REGION Network 40: *************** Alarms estop robots ***************
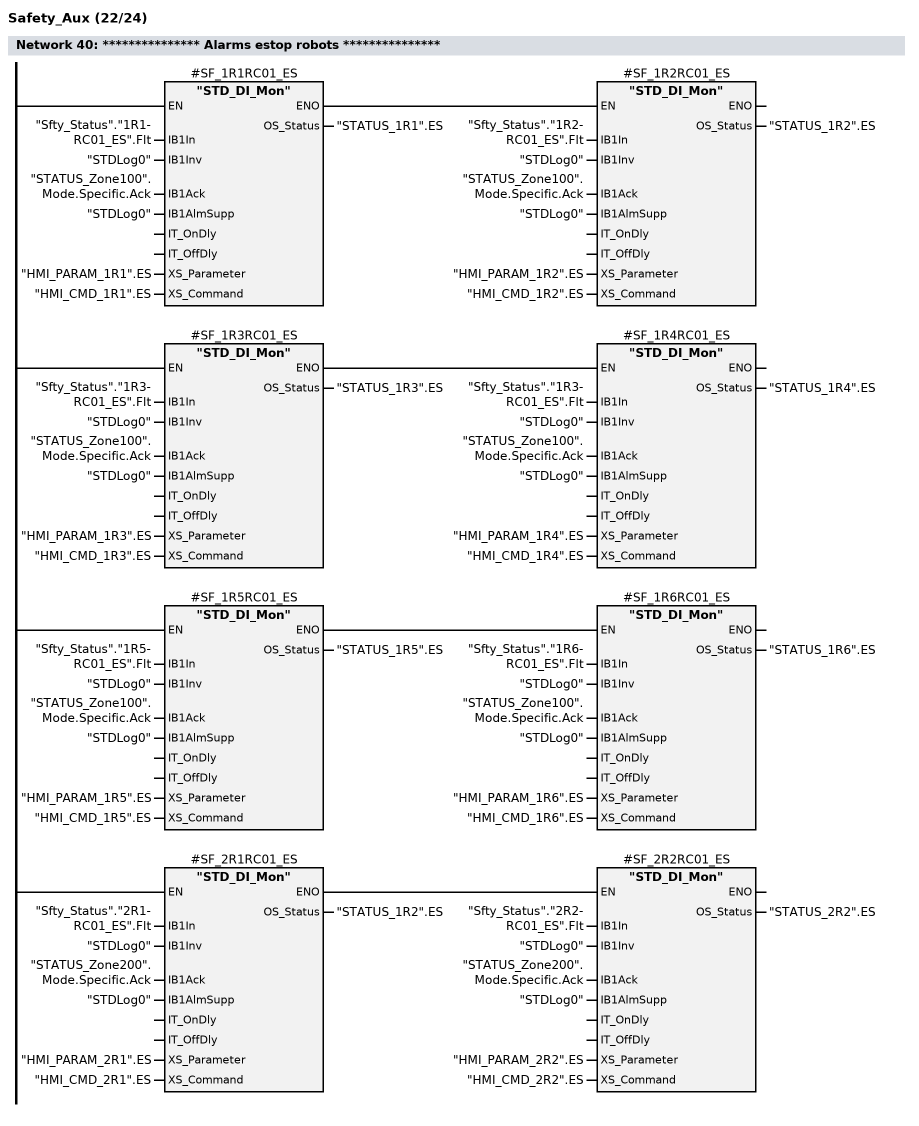
   RUNG wire#powerrail
      #SF_1R1RC01_ES(IB1In := "Sfty_Status"."1R1-RC01_ES".Flt, IB1Inv := "STDLog0", IB1Ack := "STATUS_Zone100".Mode.Specific.Ack, IB1AlmSupp := "STDLog0", IT_OnDly :=, IT_OffDly :=, XS_Parameter := "HMI_PARAM_1R1".ES, XS_Command := "HMI_CMD_1R1".ES, OS_Status => "STATUS_1R1".ES)
      #SF_1R2RC01_ES(IB1In := "Sfty_Status"."1R2-RC01_ES".Flt, IB1Inv := "STDLog0", IB1Ack := "STATUS_Zone100".Mode.Specific.Ack, IB1AlmSupp := "STDLog0", IT_OnDly :=, IT_OffDly :=, XS_Parameter := "HMI_PARAM_1R2".ES, XS_Command := "HMI_CMD_1R2".ES, OS_Status => "STATUS_1R2".ES)
   END_RUNG
   RUNG wire#powerrail
      #SF_1R3RC01_ES(IB1In := "Sfty_Status"."1R3-RC01_ES".Flt, IB1Inv := "STDLog0", IB1Ack := "STATUS_Zone100".Mode.Specific.Ack, IB1AlmSupp := "STDLog0", IT_OnDly :=, IT_OffDly :=, XS_Parameter := "HMI_PARAM_1R3".ES, XS_Command := "HMI_CMD_1R3".ES, OS_Status => "STATUS_1R3".ES)
      #SF_1R4RC01_ES(IB1In := "Sfty_Status"."1R3-RC01_ES".Flt, IB1Inv := "STDLog0", IB1Ack := "STATUS_Zone100".Mode.Specific.Ack, IB1AlmSupp := "STDLog0", IT_OnDly :=, IT_OffDly :=, XS_Parameter := "HMI_PARAM_1R4".ES, XS_Command := "HMI_CMD_1R4".ES, OS_Status => "STATUS_1R4".ES)
   END_RUNG
   RUNG wire#powerrail
      #SF_1R5RC01_ES(IB1In := "Sfty_Status"."1R5-RC01_ES".Flt, IB1Inv := "STDLog0", IB1Ack := "STATUS_Zone100".Mode.Specific.Ack, IB1AlmSupp := "STDLog0", IT_OnDly :=, IT_OffDly :=, XS_Parameter := "HMI_PARAM_1R5".ES, XS_Command := "HMI_CMD_1R5".ES, OS_Status => "STATUS_1R5".ES)
      #SF_1R6RC01_ES(IB1In := "Sfty_Status"."1R6-RC01_ES".Flt, IB1Inv := "STDLog0", IB1Ack := "STATUS_Zone100".Mode.Specific.Ack, IB1AlmSupp := "STDLog0", IT_OnDly :=, IT_OffDly :=, XS_Parameter := "HMI_PARAM_1R6".ES, XS_Command := "HMI_CMD_1R6".ES, OS_Status => "STATUS_1R6".ES)
   END_RUNG
   RUNG wire#powerrail
      #SF_2R1RC01_ES(IB1In := "Sfty_Status"."2R1-RC01_ES".Flt, IB1Inv := "STDLog0", IB1Ack := "STATUS_Zone200".Mode.Specific.Ack, IB1AlmSupp := "STDLog0", IT_OnDly :=, IT_OffDly :=, XS_Parameter := "HMI_PARAM_2R1".ES, XS_Command := "HMI_CMD_2R1".ES, OS_Status => "STATUS_1R2".ES)
      #SF_2R2RC01_ES(IB1In := "Sfty_Status"."2R2-RC01_ES".Flt, IB1Inv := "STDLog0", IB1Ack := "STATUS_Zone200".Mode.Specific.Ack, IB1AlmSupp := "STDLog0", IT_OnDly :=, IT_OffDly :=, XS_Parameter := "HMI_PARAM_2R2".ES, XS_Command := "HMI_CMD_2R2".ES, OS_Status => "STATUS_2R2".ES)
   END_RUNG
   // the same network as SCL:
   #SF_1R1RC01_ES(IB1In := "Sfty_Status"."1R1-RC01_ES".Flt,   // "STD_DI_Mon"
                  IB1Inv := "STDLog0",
                  IB1Ack := "STATUS_Zone100".Mode.Specific.Ack,
                  IB1AlmSupp := "STDLog0",
                  XS_Parameter := "HMI_PARAM_1R1".ES,
                  XS_Command := "HMI_CMD_1R1".ES,
                  OS_Status => "STATUS_1R1".ES,
                  ENO => #_w1);
   IF #_w1 THEN
       #SF_1R2RC01_ES(IB1In := "Sfty_Status"."1R2-RC01_ES".Flt,   // "STD_DI_Mon"
                      IB1Inv := "STDLog0",
                      IB1Ack := "STATUS_Zone100".Mode.Specific.Ack,
                      IB1AlmSupp := "STDLog0",
                      XS_Parameter := "HMI_PARAM_1R2".ES,
                      XS_Command := "HMI_CMD_1R2".ES,
                      OS_Status => "STATUS_1R2".ES);
   END_IF;
   #SF_1R3RC01_ES(IB1In := "Sfty_Status"."1R3-RC01_ES".Flt,   // "STD_DI_Mon"
                  IB1Inv := "STDLog0",
                  IB1Ack := "STATUS_Zone100".Mode.Specific.Ack,
                  IB1AlmSupp := "STDLog0",
                  XS_Parameter := "HMI_PARAM_1R3".ES,
                  XS_Command := "HMI_CMD_1R3".ES,
                  OS_Status => "STATUS_1R3".ES,
                  ENO => #_w2);
   IF #_w2 THEN
       #SF_1R4RC01_ES(IB1In := "Sfty_Status"."1R3-RC01_ES".Flt,   // "STD_DI_Mon"
                      IB1Inv := "STDLog0",
                      IB1Ack := "STATUS_Zone100".Mode.Specific.Ack,
                      IB1AlmSupp := "STDLog0",
                      XS_Parameter := "HMI_PARAM_1R4".ES,
                      XS_Command := "HMI_CMD_1R4".ES,
                      OS_Status => "STATUS_1R4".ES);
   END_IF;
   #SF_1R5RC01_ES(IB1In := "Sfty_Status"."1R5-RC01_ES".Flt,   // "STD_DI_Mon"
                  IB1Inv := "STDLog0",
                  IB1Ack := "STATUS_Zone100".Mode.Specific.Ack,
                  IB1AlmSupp := "STDLog0",
                  XS_Parameter := "HMI_PARAM_1R5".ES,
                  XS_Command := "HMI_CMD_1R5".ES,
                  OS_Status => "STATUS_1R5".ES,
                  ENO => #_w3);
   IF #_w3 THEN
       #SF_1R6RC01_ES(IB1In := "Sfty_Status"."1R6-RC01_ES".Flt,   // "STD_DI_Mon"
                      IB1Inv := "STDLog0",
                      IB1Ack := "STATUS_Zone100".Mode.Specific.Ack,
                      IB1AlmSupp := "STDLog0",
                      XS_Parameter := "HMI_PARAM_1R6".ES,
                      XS_Command := "HMI_CMD_1R6".ES,
                      OS_Status => "STATUS_1R6".ES);
   END_IF;
   #SF_2R1RC01_ES(IB1In := "Sfty_Status"."2R1-RC01_ES".Flt,   // "STD_DI_Mon"
                  IB1Inv := "STDLog0",
                  IB1Ack := "STATUS_Zone200".Mode.Specific.Ack,
                  IB1AlmSupp := "STDLog0",
                  XS_Parameter := "HMI_PARAM_2R1".ES,
                  XS_Command := "HMI_CMD_2R1".ES,
                  OS_Status => "STATUS_1R2".ES,
                  ENO => #_w4);
   IF #_w4 THEN
       #SF_2R2RC01_ES(IB1In := "Sfty_Status"."2R2-RC01_ES".Flt,   // "STD_DI_Mon"
                      IB1Inv := "STDLog0",
                      IB1Ack := "STATUS_Zone200".Mode.Specific.Ack,
                      IB1AlmSupp := "STDLog0",
                      XS_Parameter := "HMI_PARAM_2R2".ES,
                      XS_Command := "HMI_CMD_2R2".ES,
                      OS_Status => "STATUS_2R2".ES);
   END_IF;
END_REGION

REGION Network 41: *************** Alarms modules ***************
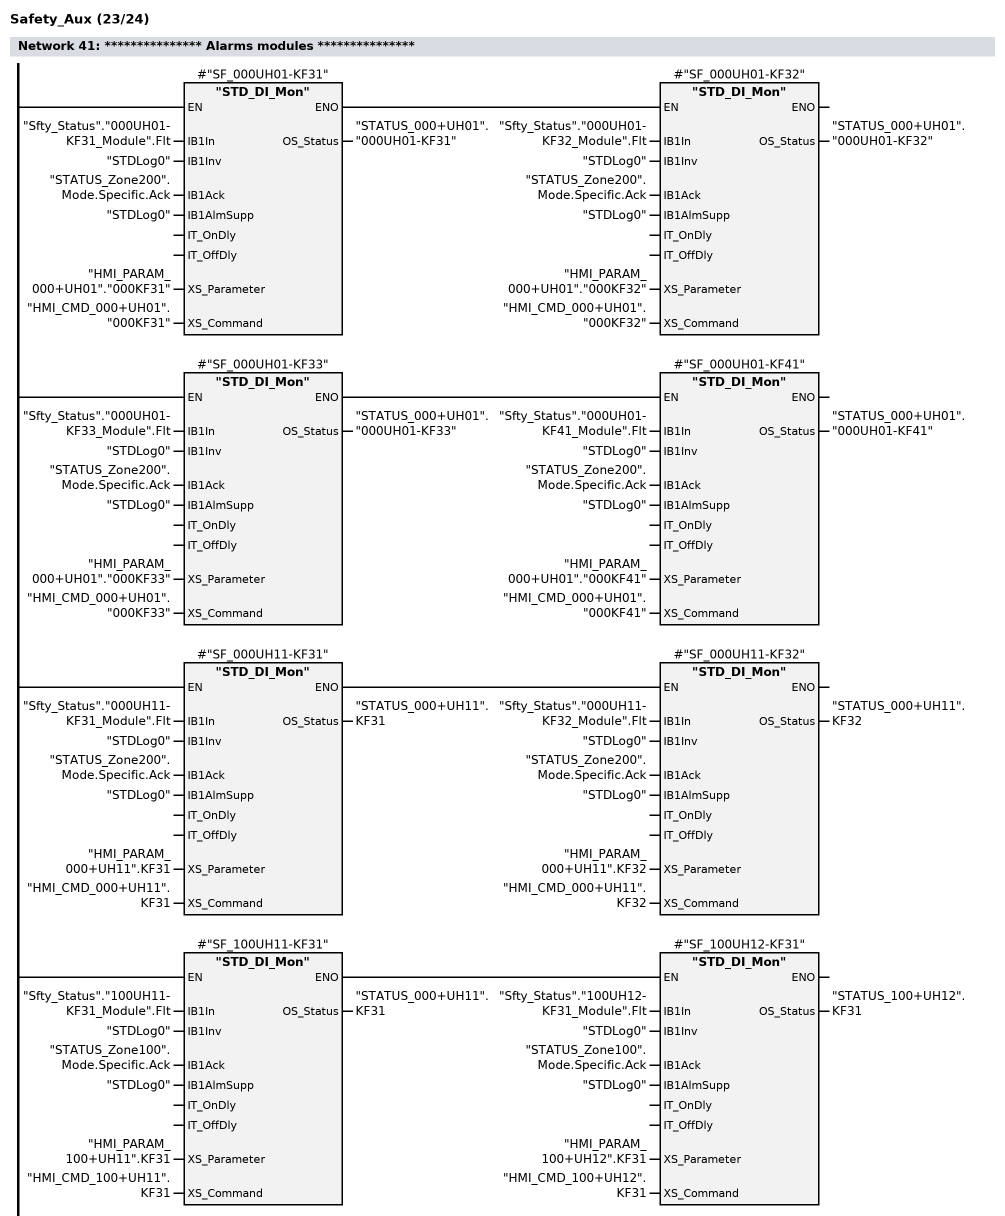
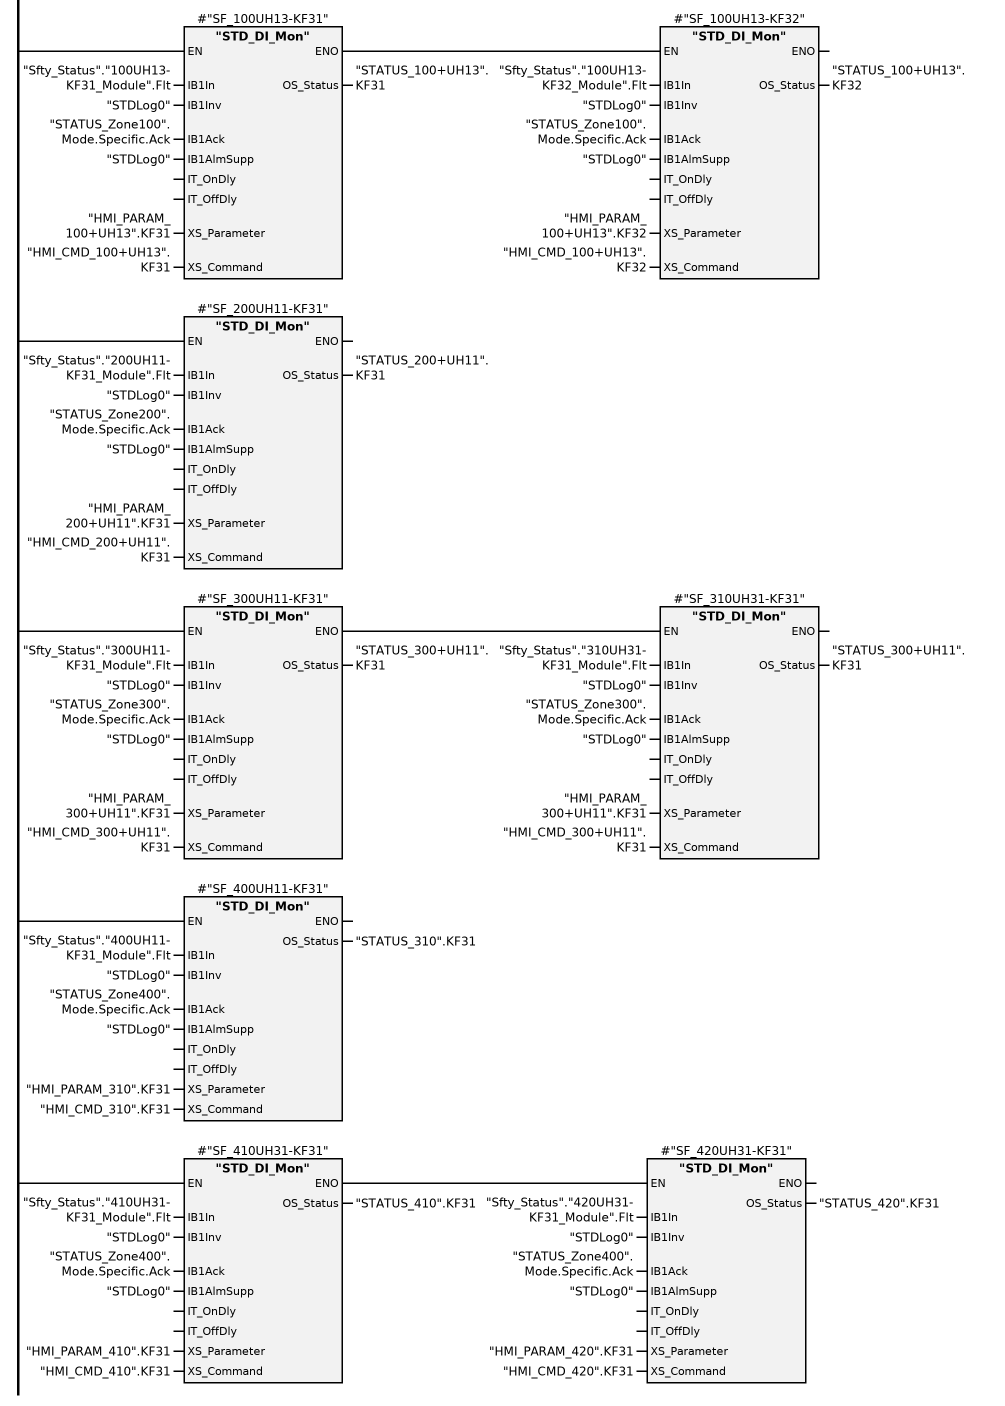
   RUNG wire#powerrail
      #"SF_000UH01-KF31"(IB1In := "Sfty_Status"."000UH01-KF31_Module".Flt, IB1Inv := "STDLog0", IB1Ack := "STATUS_Zone200".Mode.Specific.Ack, IB1AlmSupp := "STDLog0", IT_OnDly :=, IT_OffDly :=, XS_Parameter := "HMI_PARAM_000+UH01"."000KF31", XS_Command := "HMI_CMD_000+UH01"."000KF31", OS_Status => "STATUS_000+UH01"."000UH01-KF31")
      #"SF_000UH01-KF32"(IB1In := "Sfty_Status"."000UH01-KF32_Module".Flt, IB1Inv := "STDLog0", IB1Ack := "STATUS_Zone200".Mode.Specific.Ack, IB1AlmSupp := "STDLog0", IT_OnDly :=, IT_OffDly :=, XS_Parameter := "HMI_PARAM_000+UH01"."000KF32", XS_Command := "HMI_CMD_000+UH01"."000KF32", OS_Status => "STATUS_000+UH01"."000UH01-KF32")
   END_RUNG
   RUNG wire#powerrail
      #"SF_000UH01-KF33"(IB1In := "Sfty_Status"."000UH01-KF33_Module".Flt, IB1Inv := "STDLog0", IB1Ack := "STATUS_Zone200".Mode.Specific.Ack, IB1AlmSupp := "STDLog0", IT_OnDly :=, IT_OffDly :=, XS_Parameter := "HMI_PARAM_000+UH01"."000KF33", XS_Command := "HMI_CMD_000+UH01"."000KF33", OS_Status => "STATUS_000+UH01"."000UH01-KF33")
      #"SF_000UH01-KF41"(IB1In := "Sfty_Status"."000UH01-KF41_Module".Flt, IB1Inv := "STDLog0", IB1Ack := "STATUS_Zone200".Mode.Specific.Ack, IB1AlmSupp := "STDLog0", IT_OnDly :=, IT_OffDly :=, XS_Parameter := "HMI_PARAM_000+UH01"."000KF41", XS_Command := "HMI_CMD_000+UH01"."000KF41", OS_Status => "STATUS_000+UH01"."000UH01-KF41")
   END_RUNG
   RUNG wire#powerrail
      #"SF_000UH11-KF31"(IB1In := "Sfty_Status"."000UH11-KF31_Module".Flt, IB1Inv := "STDLog0", IB1Ack := "STATUS_Zone200".Mode.Specific.Ack, IB1AlmSupp := "STDLog0", IT_OnDly :=, IT_OffDly :=, XS_Parameter := "HMI_PARAM_000+UH11".KF31, XS_Command := "HMI_CMD_000+UH11".KF31, OS_Status => "STATUS_000+UH11".KF31)
      #"SF_000UH11-KF32"(IB1In := "Sfty_Status"."000UH11-KF32_Module".Flt, IB1Inv := "STDLog0", IB1Ack := "STATUS_Zone200".Mode.Specific.Ack, IB1AlmSupp := "STDLog0", IT_OnDly :=, IT_OffDly :=, XS_Parameter := "HMI_PARAM_000+UH11".KF32, XS_Command := "HMI_CMD_000+UH11".KF32, OS_Status => "STATUS_000+UH11".KF32)
   END_RUNG
   RUNG wire#powerrail
      #"SF_100UH11-KF31"(IB1In := "Sfty_Status"."100UH11-KF31_Module".Flt, IB1Inv := "STDLog0", IB1Ack := "STATUS_Zone100".Mode.Specific.Ack, IB1AlmSupp := "STDLog0", IT_OnDly :=, IT_OffDly :=, XS_Parameter := "HMI_PARAM_100+UH11".KF31, XS_Command := "HMI_CMD_100+UH11".KF31, OS_Status => "STATUS_000+UH11".KF31)
      #"SF_100UH12-KF31"(IB1In := "Sfty_Status"."100UH12-KF31_Module".Flt, IB1Inv := "STDLog0", IB1Ack := "STATUS_Zone100".Mode.Specific.Ack, IB1AlmSupp := "STDLog0", IT_OnDly :=, IT_OffDly :=, XS_Parameter := "HMI_PARAM_100+UH12".KF31, XS_Command := "HMI_CMD_100+UH12".KF31, OS_Status => "STATUS_100+UH12".KF31)
   END_RUNG
   RUNG wire#powerrail
      #"SF_100UH13-KF31"(IB1In := "Sfty_Status"."100UH13-KF31_Module".Flt, IB1Inv := "STDLog0", IB1Ack := "STATUS_Zone100".Mode.Specific.Ack, IB1AlmSupp := "STDLog0", IT_OnDly :=, IT_OffDly :=, XS_Parameter := "HMI_PARAM_100+UH13".KF31, XS_Command := "HMI_CMD_100+UH13".KF31, OS_Status => "STATUS_100+UH13".KF31)
      #"SF_100UH13-KF32"(IB1In := "Sfty_Status"."100UH13-KF32_Module".Flt, IB1Inv := "STDLog0", IB1Ack := "STATUS_Zone100".Mode.Specific.Ack, IB1AlmSupp := "STDLog0", IT_OnDly :=, IT_OffDly :=, XS_Parameter := "HMI_PARAM_100+UH13".KF32, XS_Command := "HMI_CMD_100+UH13".KF32, OS_Status => "STATUS_100+UH13".KF32)
   END_RUNG
   RUNG wire#powerrail
      #"SF_200UH11-KF31"(IB1In := "Sfty_Status"."200UH11-KF31_Module".Flt, IB1Inv := "STDLog0", IB1Ack := "STATUS_Zone200".Mode.Specific.Ack, IB1AlmSupp := "STDLog0", IT_OnDly :=, IT_OffDly :=, XS_Parameter := "HMI_PARAM_200+UH11".KF31, XS_Command := "HMI_CMD_200+UH11".KF31, OS_Status => "STATUS_200+UH11".KF31)
   END_RUNG
   RUNG wire#powerrail
      #"SF_300UH11-KF31"(IB1In := "Sfty_Status"."300UH11-KF31_Module".Flt, IB1Inv := "STDLog0", IB1Ack := "STATUS_Zone300".Mode.Specific.Ack, IB1AlmSupp := "STDLog0", IT_OnDly :=, IT_OffDly :=, XS_Parameter := "HMI_PARAM_300+UH11".KF31, XS_Command := "HMI_CMD_300+UH11".KF31, OS_Status => "STATUS_300+UH11".KF31)
      #"SF_310UH31-KF31"(IB1In := "Sfty_Status"."310UH31-KF31_Module".Flt, IB1Inv := "STDLog0", IB1Ack := "STATUS_Zone300".Mode.Specific.Ack, IB1AlmSupp := "STDLog0", IT_OnDly :=, IT_OffDly :=, XS_Parameter := "HMI_PARAM_300+UH11".KF31, XS_Command := "HMI_CMD_300+UH11".KF31, OS_Status => "STATUS_300+UH11".KF31)
   END_RUNG
   RUNG wire#powerrail
      #"SF_400UH11-KF31"(IB1In := "Sfty_Status"."400UH11-KF31_Module".Flt, IB1Inv := "STDLog0", IB1Ack := "STATUS_Zone400".Mode.Specific.Ack, IB1AlmSupp := "STDLog0", IT_OnDly :=, IT_OffDly :=, XS_Parameter := "HMI_PARAM_310".KF31, XS_Command := "HMI_CMD_310".KF31, OS_Status => "STATUS_310".KF31)
   END_RUNG
   RUNG wire#powerrail
      #"SF_410UH31-KF31"(IB1In := "Sfty_Status"."410UH31-KF31_Module".Flt, IB1Inv := "STDLog0", IB1Ack := "STATUS_Zone400".Mode.Specific.Ack, IB1AlmSupp := "STDLog0", IT_OnDly :=, IT_OffDly :=, XS_Parameter := "HMI_PARAM_410".KF31, XS_Command := "HMI_CMD_410".KF31, OS_Status => "STATUS_410".KF31)
      #"SF_420UH31-KF31"(IB1In := "Sfty_Status"."420UH31-KF31_Module".Flt, IB1Inv := "STDLog0", IB1Ack := "STATUS_Zone400".Mode.Specific.Ack, IB1AlmSupp := "STDLog0", IT_OnDly :=, IT_OffDly :=, XS_Parameter := "HMI_PARAM_420".KF31, XS_Command := "HMI_CMD_420".KF31, OS_Status => "STATUS_420".KF31)
   END_RUNG
   // the same network as SCL:
   #"SF_000UH01-KF31"(IB1In := "Sfty_Status"."000UH01-KF31_Module".Flt,   // "STD_DI_Mon"
                      IB1Inv := "STDLog0",
                      IB1Ack := "STATUS_Zone200".Mode.Specific.Ack,
                      IB1AlmSupp := "STDLog0",
                      XS_Parameter := "HMI_PARAM_000+UH01"."000KF31",
                      XS_Command := "HMI_CMD_000+UH01"."000KF31",
                      OS_Status => "STATUS_000+UH01"."000UH01-KF31",
                      ENO => #_w1);
   IF #_w1 THEN
       #"SF_000UH01-KF32"(IB1In := "Sfty_Status"."000UH01-KF32_Module".Flt,   // "STD_DI_Mon"
                          IB1Inv := "STDLog0",
                          IB1Ack := "STATUS_Zone200".Mode.Specific.Ack,
                          IB1AlmSupp := "STDLog0",
                          XS_Parameter := "HMI_PARAM_000+UH01"."000KF32",
                          XS_Command := "HMI_CMD_000+UH01"."000KF32",
                          OS_Status => "STATUS_000+UH01"."000UH01-KF32");
   END_IF;
   #"SF_000UH01-KF33"(IB1In := "Sfty_Status"."000UH01-KF33_Module".Flt,   // "STD_DI_Mon"
                      IB1Inv := "STDLog0",
                      IB1Ack := "STATUS_Zone200".Mode.Specific.Ack,
                      IB1AlmSupp := "STDLog0",
                      XS_Parameter := "HMI_PARAM_000+UH01"."000KF33",
                      XS_Command := "HMI_CMD_000+UH01"."000KF33",
                      OS_Status => "STATUS_000+UH01"."000UH01-KF33",
                      ENO => #_w2);
   IF #_w2 THEN
       #"SF_000UH01-KF41"(IB1In := "Sfty_Status"."000UH01-KF41_Module".Flt,   // "STD_DI_Mon"
                          IB1Inv := "STDLog0",
                          IB1Ack := "STATUS_Zone200".Mode.Specific.Ack,
                          IB1AlmSupp := "STDLog0",
                          XS_Parameter := "HMI_PARAM_000+UH01"."000KF41",
                          XS_Command := "HMI_CMD_000+UH01"."000KF41",
                          OS_Status => "STATUS_000+UH01"."000UH01-KF41");
   END_IF;
   #"SF_000UH11-KF31"(IB1In := "Sfty_Status"."000UH11-KF31_Module".Flt,   // "STD_DI_Mon"
                      IB1Inv := "STDLog0",
                      IB1Ack := "STATUS_Zone200".Mode.Specific.Ack,
                      IB1AlmSupp := "STDLog0",
                      XS_Parameter := "HMI_PARAM_000+UH11".KF31,
                      XS_Command := "HMI_CMD_000+UH11".KF31,
                      OS_Status => "STATUS_000+UH11".KF31,
                      ENO => #_w3);
   IF #_w3 THEN
       #"SF_000UH11-KF32"(IB1In := "Sfty_Status"."000UH11-KF32_Module".Flt,   // "STD_DI_Mon"
                          IB1Inv := "STDLog0",
                          IB1Ack := "STATUS_Zone200".Mode.Specific.Ack,
                          IB1AlmSupp := "STDLog0",
                          XS_Parameter := "HMI_PARAM_000+UH11".KF32,
                          XS_Command := "HMI_CMD_000+UH11".KF32,
                          OS_Status => "STATUS_000+UH11".KF32);
   END_IF;
   #"SF_100UH11-KF31"(IB1In := "Sfty_Status"."100UH11-KF31_Module".Flt,   // "STD_DI_Mon"
                      IB1Inv := "STDLog0",
                      IB1Ack := "STATUS_Zone100".Mode.Specific.Ack,
                      IB1AlmSupp := "STDLog0",
                      XS_Parameter := "HMI_PARAM_100+UH11".KF31,
                      XS_Command := "HMI_CMD_100+UH11".KF31,
                      OS_Status => "STATUS_000+UH11".KF31,
                      ENO => #_w4);
   IF #_w4 THEN
       #"SF_100UH12-KF31"(IB1In := "Sfty_Status"."100UH12-KF31_Module".Flt,   // "STD_DI_Mon"
                          IB1Inv := "STDLog0",
                          IB1Ack := "STATUS_Zone100".Mode.Specific.Ack,
                          IB1AlmSupp := "STDLog0",
                          XS_Parameter := "HMI_PARAM_100+UH12".KF31,
                          XS_Command := "HMI_CMD_100+UH12".KF31,
                          OS_Status => "STATUS_100+UH12".KF31);
   END_IF;
   #"SF_100UH13-KF31"(IB1In := "Sfty_Status"."100UH13-KF31_Module".Flt,   // "STD_DI_Mon"
                      IB1Inv := "STDLog0",
                      IB1Ack := "STATUS_Zone100".Mode.Specific.Ack,
                      IB1AlmSupp := "STDLog0",
                      XS_Parameter := "HMI_PARAM_100+UH13".KF31,
                      XS_Command := "HMI_CMD_100+UH13".KF31,
                      OS_Status => "STATUS_100+UH13".KF31,
                      ENO => #_w5);
   IF #_w5 THEN
       #"SF_100UH13-KF32"(IB1In := "Sfty_Status"."100UH13-KF32_Module".Flt,   // "STD_DI_Mon"
                          IB1Inv := "STDLog0",
                          IB1Ack := "STATUS_Zone100".Mode.Specific.Ack,
                          IB1AlmSupp := "STDLog0",
                          XS_Parameter := "HMI_PARAM_100+UH13".KF32,
                          XS_Command := "HMI_CMD_100+UH13".KF32,
                          OS_Status => "STATUS_100+UH13".KF32);
   END_IF;
   #"SF_200UH11-KF31"(IB1In := "Sfty_Status"."200UH11-KF31_Module".Flt,   // "STD_DI_Mon"
                      IB1Inv := "STDLog0",
                      IB1Ack := "STATUS_Zone200".Mode.Specific.Ack,
                      IB1AlmSupp := "STDLog0",
                      XS_Parameter := "HMI_PARAM_200+UH11".KF31,
                      XS_Command := "HMI_CMD_200+UH11".KF31,
                      OS_Status => "STATUS_200+UH11".KF31);
   #"SF_300UH11-KF31"(IB1In := "Sfty_Status"."300UH11-KF31_Module".Flt,   // "STD_DI_Mon"
                      IB1Inv := "STDLog0",
                      IB1Ack := "STATUS_Zone300".Mode.Specific.Ack,
                      IB1AlmSupp := "STDLog0",
                      XS_Parameter := "HMI_PARAM_300+UH11".KF31,
                      XS_Command := "HMI_CMD_300+UH11".KF31,
                      OS_Status => "STATUS_300+UH11".KF31,
                      ENO => #_w6);
   IF #_w6 THEN
       #"SF_310UH31-KF31"(IB1In := "Sfty_Status"."310UH31-KF31_Module".Flt,   // "STD_DI_Mon"
                          IB1Inv := "STDLog0",
                          IB1Ack := "STATUS_Zone300".Mode.Specific.Ack,
                          IB1AlmSupp := "STDLog0",
                          XS_Parameter := "HMI_PARAM_300+UH11".KF31,
                          XS_Command := "HMI_CMD_300+UH11".KF31,
                          OS_Status => "STATUS_300+UH11".KF31);
   END_IF;
   #"SF_400UH11-KF31"(IB1In := "Sfty_Status"."400UH11-KF31_Module".Flt,   // "STD_DI_Mon"
                      IB1Inv := "STDLog0",
                      IB1Ack := "STATUS_Zone400".Mode.Specific.Ack,
                      IB1AlmSupp := "STDLog0",
                      XS_Parameter := "HMI_PARAM_310".KF31,
                      XS_Command := "HMI_CMD_310".KF31,
                      OS_Status => "STATUS_310".KF31);
   #"SF_410UH31-KF31"(IB1In := "Sfty_Status"."410UH31-KF31_Module".Flt,   // "STD_DI_Mon"
                      IB1Inv := "STDLog0",
                      IB1Ack := "STATUS_Zone400".Mode.Specific.Ack,
                      IB1AlmSupp := "STDLog0",
                      XS_Parameter := "HMI_PARAM_410".KF31,
                      XS_Command := "HMI_CMD_410".KF31,
                      OS_Status => "STATUS_410".KF31,
                      ENO => #_w7);
   IF #_w7 THEN
       #"SF_420UH31-KF31"(IB1In := "Sfty_Status"."420UH31-KF31_Module".Flt,   // "STD_DI_Mon"
                          IB1Inv := "STDLog0",
                          IB1Ack := "STATUS_Zone400".Mode.Specific.Ack,
                          IB1AlmSupp := "STDLog0",
                          XS_Parameter := "HMI_PARAM_420".KF31,
                          XS_Command := "HMI_CMD_420".KF31,
                          OS_Status => "STATUS_420".KF31);
   END_IF;
END_REGION

REGION Network 42: *************** Alarms gate module ***************
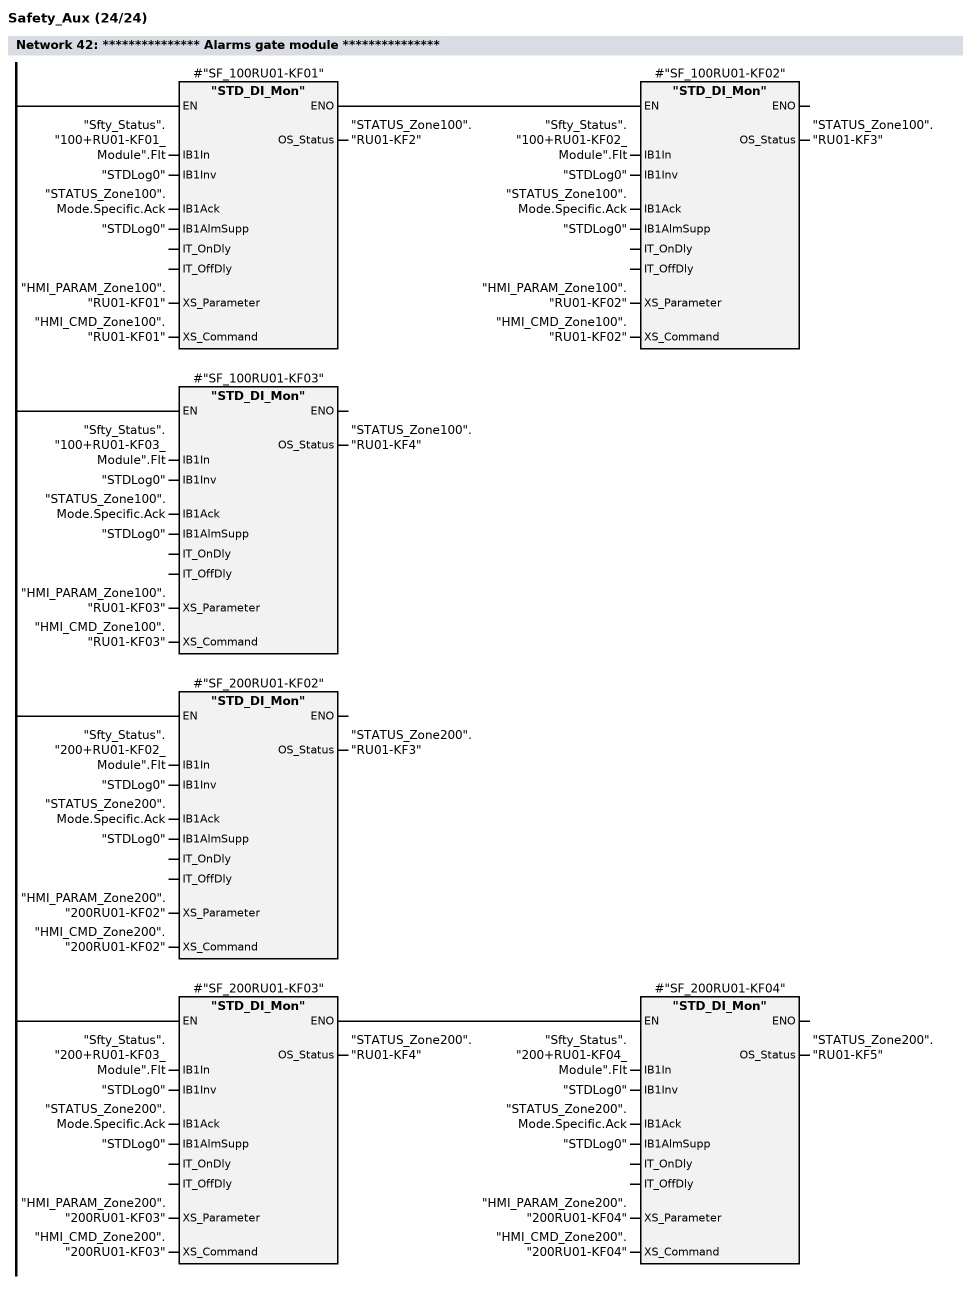
   RUNG wire#powerrail
      #"SF_100RU01-KF01"(IB1In := "Sfty_Status"."100+RU01-KF01_Module".Flt, IB1Inv := "STDLog0", IB1Ack := "STATUS_Zone100".Mode.Specific.Ack, IB1AlmSupp := "STDLog0", IT_OnDly :=, IT_OffDly :=, XS_Parameter := "HMI_PARAM_Zone100"."RU01-KF01", XS_Command := "HMI_CMD_Zone100"."RU01-KF01", OS_Status => "STATUS_Zone100"."RU01-KF2")
      #"SF_100RU01-KF02"(IB1In := "Sfty_Status"."100+RU01-KF02_Module".Flt, IB1Inv := "STDLog0", IB1Ack := "STATUS_Zone100".Mode.Specific.Ack, IB1AlmSupp := "STDLog0", IT_OnDly :=, IT_OffDly :=, XS_Parameter := "HMI_PARAM_Zone100"."RU01-KF02", XS_Command := "HMI_CMD_Zone100"."RU01-KF02", OS_Status => "STATUS_Zone100"."RU01-KF3")
   END_RUNG
   RUNG wire#powerrail
      #"SF_100RU01-KF03"(IB1In := "Sfty_Status"."100+RU01-KF03_Module".Flt, IB1Inv := "STDLog0", IB1Ack := "STATUS_Zone100".Mode.Specific.Ack, IB1AlmSupp := "STDLog0", IT_OnDly :=, IT_OffDly :=, XS_Parameter := "HMI_PARAM_Zone100"."RU01-KF03", XS_Command := "HMI_CMD_Zone100"."RU01-KF03", OS_Status => "STATUS_Zone100"."RU01-KF4")
   END_RUNG
   RUNG wire#powerrail
      #"SF_200RU01-KF02"(IB1In := "Sfty_Status"."200+RU01-KF02_Module".Flt, IB1Inv := "STDLog0", IB1Ack := "STATUS_Zone200".Mode.Specific.Ack, IB1AlmSupp := "STDLog0", IT_OnDly :=, IT_OffDly :=, XS_Parameter := "HMI_PARAM_Zone200"."200RU01-KF02", XS_Command := "HMI_CMD_Zone200"."200RU01-KF02", OS_Status => "STATUS_Zone200"."RU01-KF3")
   END_RUNG
   RUNG wire#powerrail
      #"SF_200RU01-KF03"(IB1In := "Sfty_Status"."200+RU01-KF03_Module".Flt, IB1Inv := "STDLog0", IB1Ack := "STATUS_Zone200".Mode.Specific.Ack, IB1AlmSupp := "STDLog0", IT_OnDly :=, IT_OffDly :=, XS_Parameter := "HMI_PARAM_Zone200"."200RU01-KF03", XS_Command := "HMI_CMD_Zone200"."200RU01-KF03", OS_Status => "STATUS_Zone200"."RU01-KF4")
      #"SF_200RU01-KF04"(IB1In := "Sfty_Status"."200+RU01-KF04_Module".Flt, IB1Inv := "STDLog0", IB1Ack := "STATUS_Zone200".Mode.Specific.Ack, IB1AlmSupp := "STDLog0", IT_OnDly :=, IT_OffDly :=, XS_Parameter := "HMI_PARAM_Zone200"."200RU01-KF04", XS_Command := "HMI_CMD_Zone200"."200RU01-KF04", OS_Status => "STATUS_Zone200"."RU01-KF5")
   END_RUNG
   // the same network as SCL:
   #"SF_100RU01-KF01"(IB1In := "Sfty_Status"."100+RU01-KF01_Module".Flt,   // "STD_DI_Mon"
                      IB1Inv := "STDLog0",
                      IB1Ack := "STATUS_Zone100".Mode.Specific.Ack,
                      IB1AlmSupp := "STDLog0",
                      XS_Parameter := "HMI_PARAM_Zone100"."RU01-KF01",
                      XS_Command := "HMI_CMD_Zone100"."RU01-KF01",
                      OS_Status => "STATUS_Zone100"."RU01-KF2",
                      ENO => #_w1);
   IF #_w1 THEN
       #"SF_100RU01-KF02"(IB1In := "Sfty_Status"."100+RU01-KF02_Module".Flt,   // "STD_DI_Mon"
                          IB1Inv := "STDLog0",
                          IB1Ack := "STATUS_Zone100".Mode.Specific.Ack,
                          IB1AlmSupp := "STDLog0",
                          XS_Parameter := "HMI_PARAM_Zone100"."RU01-KF02",
                          XS_Command := "HMI_CMD_Zone100"."RU01-KF02",
                          OS_Status => "STATUS_Zone100"."RU01-KF3");
   END_IF;
   #"SF_100RU01-KF03"(IB1In := "Sfty_Status"."100+RU01-KF03_Module".Flt,   // "STD_DI_Mon"
                      IB1Inv := "STDLog0",
                      IB1Ack := "STATUS_Zone100".Mode.Specific.Ack,
                      IB1AlmSupp := "STDLog0",
                      XS_Parameter := "HMI_PARAM_Zone100"."RU01-KF03",
                      XS_Command := "HMI_CMD_Zone100"."RU01-KF03",
                      OS_Status => "STATUS_Zone100"."RU01-KF4");
   #"SF_200RU01-KF02"(IB1In := "Sfty_Status"."200+RU01-KF02_Module".Flt,   // "STD_DI_Mon"
                      IB1Inv := "STDLog0",
                      IB1Ack := "STATUS_Zone200".Mode.Specific.Ack,
                      IB1AlmSupp := "STDLog0",
                      XS_Parameter := "HMI_PARAM_Zone200"."200RU01-KF02",
                      XS_Command := "HMI_CMD_Zone200"."200RU01-KF02",
                      OS_Status => "STATUS_Zone200"."RU01-KF3");
   #"SF_200RU01-KF03"(IB1In := "Sfty_Status"."200+RU01-KF03_Module".Flt,   // "STD_DI_Mon"
                      IB1Inv := "STDLog0",
                      IB1Ack := "STATUS_Zone200".Mode.Specific.Ack,
                      IB1AlmSupp := "STDLog0",
                      XS_Parameter := "HMI_PARAM_Zone200"."200RU01-KF03",
                      XS_Command := "HMI_CMD_Zone200"."200RU01-KF03",
                      OS_Status => "STATUS_Zone200"."RU01-KF4",
                      ENO => #_w2);
   IF #_w2 THEN
       #"SF_200RU01-KF04"(IB1In := "Sfty_Status"."200+RU01-KF04_Module".Flt,   // "STD_DI_Mon"
                          IB1Inv := "STDLog0",
                          IB1Ack := "STATUS_Zone200".Mode.Specific.Ack,
                          IB1AlmSupp := "STDLog0",
                          XS_Parameter := "HMI_PARAM_Zone200"."200RU01-KF04",
                          XS_Command := "HMI_CMD_Zone200"."200RU01-KF04",
                          OS_Status => "STATUS_Zone200"."RU01-KF5");
   END_IF;
END_REGION
END_FUNCTION_BLOCK
